Fanuc KAREL source: kt00749.KL

-- PROVISIONAL review KL for V940-1; original PC SHA256 958449f34f21858516425f7deef1aac900955e6dfe6baabaf4b32d228f68e77f
-- Incomplete behavior may be omitted. Consult companion uncertainty JSON. Do not deploy.
PROGRAM KT00749
%NOLOCKGROUP
VAR
  I1 : INTEGER
  I2 : INTEGER
  OUT : REAL
BEGIN
  -- V9_ZERO_TABLE_METADATA_HINT layout=0001; no indexed target words; source/name/runtime held
  -- UNRESOLVED_PC offsets 5-16; opcodes 2E,23
  -- UNRESOLVED_PC offsets 21-32; opcodes 2E,23
  -- UNRESOLVED_PC offsets 37-48; opcodes 2E,23
  -- UNRESOLVED_PC offsets 53-64; opcodes 2E,23
  -- UNRESOLVED_PC offsets 69-83; opcodes 21,50,64,23
  -- UNRESOLVED_PC offsets 88-92; opcodes 7F
END KT00749
